KUKA KRL program: ToolRackTest.src

&ACCESS RVP
&REL 46
&PARAM EDITMASK = *
&PARAM TEMPLATE = C:\KRC\Roboter\Template\vorgabe
DEF ToolrackTest( )
;FOLD INI;%{PE}
  ;FOLD BASISTECH INI
    GLOBAL INTERRUPT DECL 3 WHEN $STOPMESS==TRUE DO IR_STOPM ( )
    INTERRUPT ON 3
    BAS (#INITMOV,0 )
  ;ENDFOLD (BASISTECH INI)
  ;FOLD USER INI
    ;Make your modifications here

  ;ENDFOLD (USER INI)
;ENDFOLD (INI)

;************************************************
;              CNC Robotics Ltd
;              www.cncrobotics.co.uk
;************************************************
;     Contact: helpdesk@cncrobotics.co.uk
;     Date: 25/09/23
;     Version: 0.13.46
;************************************************
; Description: Program to make test each position
; of the toolrack
;************************************************

;FOR MANUAL TOOL TAKE PLEASE CHANGE THE REQUIRED TOOL NUMBER IN THE BRACKETS

CheckEOATooling(#SPINDLE)

ToolrackMove(1)
;wait sec 0.5
;ToolrackMove(2)
;wait sec 0.5
;ToolrackMove(3)
;wait sec 0.5
;ToolrackMove(4)
;wait sec 0.5
;ToolrackMove(5)
;wait sec 0.5
;ToolrackMove(6)
;wait sec 0.5
;ToolrackMove(7)
;wait sec 0.5
;ToolrackMove(8)

END
